FUNCTION_BLOCK Recipe_10021_TequilaSunrise_Alternative
VAR_INPUT
	TaskID	: 	LREAL;
	Execute :	BOOL;
	Parameter	: ARRAY [1..RecipeParameterCnt] OF DUT_RECIPE_PARAMETERINPUT;
END_VAR
VAR_OUTPUT
	RecipeDone	: BOOL;
END_VAR
VAR	
	Done		: BOOL;
	Priority	: INT;
	
END_VAR

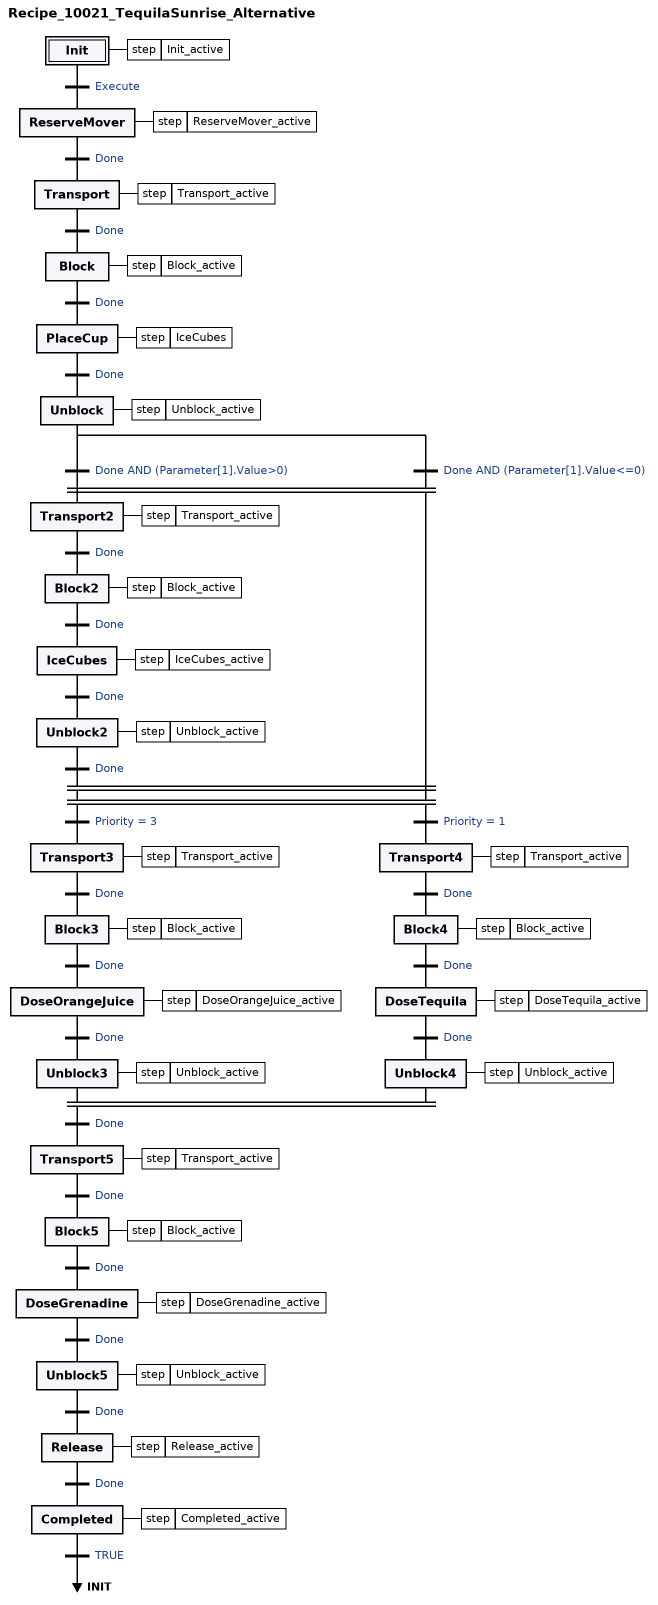
INITIAL_STEP Init:
    Init_active(N);  // step action
END_STEP
TRANSITION FROM Init TO ReserveMover
    := Execute;
END_TRANSITION
STEP ReserveMover:
    ReserveMover_active(N);  // step action
END_STEP
TRANSITION FROM ReserveMover TO Transport
    := Done;
END_TRANSITION
STEP Transport:
    Transport_active(N);  // step action
END_STEP
TRANSITION FROM Transport TO Block
    := Done;
END_TRANSITION
STEP Block:
    Block_active(N);  // step action
END_STEP
TRANSITION FROM Block TO PlaceCup
    := Done;
END_TRANSITION
STEP PlaceCup:
    IceCubes(N);  // step action
END_STEP
TRANSITION FROM PlaceCup TO Unblock
    := Done;
END_TRANSITION
STEP Unblock:
    Unblock_active(N);  // step action
END_STEP
TRANSITION FROM Unblock TO Transport2
    := Done AND (Parameter[1].Value>0);
END_TRANSITION
STEP Transport2:
    Transport_active(N);  // step action
END_STEP
TRANSITION FROM Transport2 TO Block2
    := Done;
END_TRANSITION
STEP Block2:
    Block_active(N);  // step action
END_STEP
TRANSITION FROM Block2 TO IceCubes
    := Done;
END_TRANSITION
STEP IceCubes:
    IceCubes_active(N);  // step action
END_STEP
TRANSITION FROM IceCubes TO Unblock2
    := Done;
END_TRANSITION
STEP Unblock2:
    Unblock_active(N);  // step action
END_STEP
TRANSITION FROM Unblock2 TO (???, ???)
    := Done;
END_TRANSITION
TRANSITION FROM Unblock TO (???, ???)
    := Done AND (Parameter[1].Value<=0);
END_TRANSITION
TRANSITION FROM (???, ???) TO Transport3
    := Priority = 3;
END_TRANSITION
STEP Transport3:
    Transport_active(N);  // step action
END_STEP
TRANSITION FROM Transport3 TO Block3
    := Done;
END_TRANSITION
STEP Block3:
    Block_active(N);  // step action
END_STEP
TRANSITION FROM Block3 TO DoseOrangeJuice
    := Done;
END_TRANSITION
STEP DoseOrangeJuice:
    DoseOrangeJuice_active(N);  // step action
END_STEP
TRANSITION FROM DoseOrangeJuice TO Unblock3
    := Done;
END_TRANSITION
STEP Unblock3:
    Unblock_active(N);  // step action
END_STEP
TRANSITION FROM (???, ???) TO Transport4
    := Priority = 1;
END_TRANSITION
STEP Transport4:
    Transport_active(N);  // step action
END_STEP
TRANSITION FROM Transport4 TO Block4
    := Done;
END_TRANSITION
STEP Block4:
    Block_active(N);  // step action
END_STEP
TRANSITION FROM Block4 TO DoseTequila
    := Done;
END_TRANSITION
STEP DoseTequila:
    DoseTequila_active(N);  // step action
END_STEP
TRANSITION FROM DoseTequila TO Unblock4
    := Done;
END_TRANSITION
STEP Unblock4:
    Unblock_active(N);  // step action
END_STEP
TRANSITION FROM (Unblock3, Unblock4) TO Transport5
    := Done;
END_TRANSITION
STEP Transport5:
    Transport_active(N);  // step action
END_STEP
TRANSITION FROM Transport5 TO Block5
    := Done;
END_TRANSITION
STEP Block5:
    Block_active(N);  // step action
END_STEP
TRANSITION FROM Block5 TO DoseGrenadine
    := Done;
END_TRANSITION
STEP DoseGrenadine:
    DoseGrenadine_active(N);  // step action
END_STEP
TRANSITION FROM DoseGrenadine TO Unblock5
    := Done;
END_TRANSITION
STEP Unblock5:
    Unblock_active(N);  // step action
END_STEP
TRANSITION FROM Unblock5 TO Release
    := Done;
END_TRANSITION
STEP Release:
    Release_active(N);  // step action
END_STEP
TRANSITION FROM Release TO Completed
    := Done;
END_TRANSITION
STEP Completed:
    Completed_active(N);  // step action
END_STEP
TRANSITION FROM Completed TO INIT
    := TRUE;
END_TRANSITION

ACTION Release_active:
Done := FALSE;


ExecuteSkill.SkillID 			:= 1311;
ExecuteSkill.SkillName	 		:= 'Release Mover';
ExecuteSkill.Parameter[1].ID 	:= 1;
ExecuteSkill.Parameter[1].Name 	:= 'TaskID';
ExecuteSkill.Parameter[1].Value := TaskID;
ExecuteSkill();

Done := TRUE;
END_ACTION

ACTION DoseTequila_active:
Done := FALSE;

ExecuteSkill.SkillID 			:= 1009;
ExecuteSkill.SkillName	 		:= 'Dose Tequila';
ExecuteSkill.Parameter[1].ID 	:= 1;
ExecuteSkill.Parameter[1].Name 	:= 'Amount';
ExecuteSkill.Parameter[1].Value := 50;//[ml]
ExecuteSkill();
Done := TRUE;
END_ACTION

ACTION IceCubes_active:
Done := FALSE;

ExecuteSkill.SkillID 			:= 1401;
ExecuteSkill.SkillName	 		:= 'Dispense Ice Cubes';
ExecuteSkill.Parameter[1].ID 	:= 1;
ExecuteSkill.Parameter[1].Name 	:= 'Amount';
ExecuteSkill.Parameter[1].Value := Parameter[1].Value;
ExecuteSkill();
Done := TRUE;
END_ACTION

ACTION Init_active:
RecipeDone := FALSE;
END_ACTION

ACTION DoseOrangeJuice_active:
Done := FALSE;

ExecuteSkill.SkillID 			:= 1011;
ExecuteSkill.SkillName	 		:= 'Dose Orange Juice';
ExecuteSkill.Parameter[1].ID 	:= 1;
ExecuteSkill.Parameter[1].Name 	:= 'Amount';
ExecuteSkill.Parameter[1].Value := 133;//[ml]
ExecuteSkill();
Done := TRUE;
END_ACTION

ACTION DoseGrenadine_active:
Done := FALSE;

ExecuteSkill.SkillID 			:= 1012;
ExecuteSkill.SkillName	 		:= 'Dose Orange Juice';
ExecuteSkill.Parameter[1].ID 	:= 1;
ExecuteSkill.Parameter[1].Name 	:= 'Amount';
ExecuteSkill.Parameter[1].Value := 12;//[ml]

ExecuteSkill.Parameter[2].ID 	:= 2;
ExecuteSkill.Parameter[2].Name 	:= 'SpeedFaktor';
ExecuteSkill.Parameter[2].Value := 0,5;//[ml]


ExecuteSkill();
Done := TRUE;
END_ACTION

ACTION Completed_active:
RecipeDone := TRUE;
Execute := FALSE;
Done := FALSE;
END_ACTION

ACTION ReserveMover_active:
Done := FALSE;


ExecuteSkill.SkillID := 1310;
ExecuteSkill.SkillName	 := 'Reserve Mover';
ExecuteSkill.Parameter[1].ID := 1;
ExecuteSkill.Parameter[1].Name := 'TaskID';
ExecuteSkill.Parameter[1].Value := TaskID;
ExecuteSkill();

Done := TRUE;
END_ACTION

ACTION Block_active:
Done := FALSE;

//Skill auswählen
ExecuteSkill.SkillID := 1315;
ExecuteSkill.SkillName	 := 'Block Mover';

//Parameter setzen
ExecuteSkill.Parameter[1].ID := 1;
ExecuteSkill.Parameter[1].Name := 'TaskID';
ExecuteSkill.Parameter[1].Value := TaskID;

//Skill hinzufügen
ExecuteSkill();


Done := TRUE;
END_ACTION

ACTION Transport_active:
Done := FALSE;

//Skill auswählen
ExecuteSkill.SkillID 		:= 1320;
ExecuteSkill.SkillName	 	:= 'Transport Mover';

//Geschwindigkeit setzen
ExecuteSkill.Parameter[1].ID := 3;
ExecuteSkill.Parameter[1].Name := 'Velocity';
ExecuteSkill.Parameter[1].Value := 3000;


ExecuteSkill();

Done := ExecuteSkill.Done;
END_ACTION

ACTION Unblock_active:
Done := FALSE;

//Skill auswählen
ExecuteSkill.SkillID := 1316;
ExecuteSkill.SkillName	 := 'Unblock Mover';

//Parameter setzen
ExecuteSkill.Parameter[1].ID := 1;
ExecuteSkill.Parameter[1].Name := 'TaskID';
ExecuteSkill.Parameter[1].Value := TaskID;

//Skill hinzufügen
ExecuteSkill();


Done := TRUE;
END_ACTION

ACTION IceCubes:
Done := FALSE;

ExecuteSkill.SkillID 			:= 1402;
ExecuteSkill.SkillName	 		:= 'Place Cup';

ExecuteSkill();
Done := TRUE;
END_ACTION

END_FUNCTION_BLOCK

(* stored: Version 1.1.0.1, ProductVersion 3.1.0.25
   POU Recipe_10021_TequilaSunrise_Alternative: Id {a5dbc547-6bba-4801-8d9d-8905ba9a2da8}
   Action Release_active: Id {0adf638e-9f7b-4c49-bd53-fc11ee11df23}
   Action DoseTequila_active: Id {120cf29d-dff1-42a0-8b7e-220651bd541a}
   Action IceCubes_active: Id {17b3c754-267a-4cd6-a9ed-3eb115deb612}
   Action Init_active: Id {49483e6e-b596-489a-8ff5-3c553fedb024}
   Action DoseOrangeJuice_active: Id {98f9508d-02dc-4e6a-932a-6a9272a63678}
   Action DoseGrenadine_active: Id {ae7b7187-b486-4a40-a99e-0146f020a36c}
   Action Completed_active: Id {af01477d-7cc3-4dd5-9b67-20582fd1fdff}
   Action ReserveMover_active: Id {bd286002-2148-4c1f-ba96-995717342777}
   Action Block_active: Id {c63f14ca-82cb-4959-9f75-80aa2caf467f}
   Action Transport_active: Id {d5bca688-2749-4d5c-abfa-0ec4597f7e49}
   Action Unblock_active: Id {e0c68527-b543-404a-aeaf-800f7b036a9b}
   Action IceCubes: Id {f4c054e3-b1bd-4422-bbdb-51bb8c5f1bca} *)
